(* IEC 61131-3 sources: Industry-PLC-LLM/data/PLCBEAD_repo/PLCBEAD_PLCEmbed-main/PLC-BEAD/Source/GEB/DAYS_IN_YEAR, 1 file *)

(* ---- DAYS_IN_YEAR.ST ---- *)
FUNCTION LEAP_OF_DATE:BOOL

	VAR_INPUT
		IDATE :	UDINT;
	END_VAR

	LEAP_OF_DATE := SHL(UDINT_TO_DWORD((IDATE + UDINT#43200) / UDINT#31557600), 30) = DWORD#16#80000000;
END_FUNCTION

FUNCTION DAYS_IN_YEAR:INT
	VAR_INPUT
		IDATE :	UDINT;
	END_VAR

	IF LEAP_OF_DATE(IDATE) THEN
		DAYS_IN_YEAR  := 366;
	ELSE
		DAYS_IN_YEAR  := 365;
	END_IF;
END_FUNCTION

PROGRAM program0
  VAR
    LocalVar0 : UDINT;
	LocalOUT  : INT;
  END_VAR
  	LocalOUT := DAYS_IN_YEAR(LocalVar0);
END_PROGRAM
